/// <summary>
/// Two-Way-Actuator analog (mixing valve)
/// Zwei-Wege-Stellglied analog (Mischventil)
/// </summary>
FUNCTION_BLOCK PAEActuator2way_Analog EXTENDS PAEActuator1way_Analog
VAR_INPUT
	_IPos2 AT %I*: BOOL;	
END_VAR
VAR_OUTPUT
	_QPos2 AT %Q*: BOOL;	
END_VAR
VAR
	_PAPointMatIn2  : PAPoint(THIS^);
END_VAR

METHOD FB_init : BOOL
VAR_INPUT
	bInitRetains : BOOL; // if TRUE, the retain variables are initialized (warm start / cold start)
	bInCopyCode : BOOL;  // if TRUE, the instance afterwards gets moved into the copy code (online change)
	parent : IACComponent;
END_VAR
AddPoint(_PAPointMatIn1);
END_METHOD

METHOD PUBLIC HasPointReachedOffPosition : BOOL
VAR_INPUT
	point : IACPoint;
END_VAR
HasPointReachedOffPosition := SUPER^.HasPointReachedOffPosition(point);
END_METHOD

METHOD PUBLIC HasPointReachedOnPosition : BOOL
VAR_INPUT
	point : IACPoint;
END_VAR
HasPointReachedOnPosition := SUPER^.HasPointReachedOnPosition(point);
END_METHOD

PROPERTY PUBLIC PAPointMatIn2 : IACPoint
GET
PAPointMatIn2  := _PAPointMatIn2;
END_GET
END_PROPERTY

END_FUNCTION_BLOCK

(* stored: Version 1.1.0.1, ProductVersion 3.1.4020.12
   POU PAEActuator2way_Analog: Id {a2a041d8-6df1-467d-bb65-37358f54a768}, SpecialFunc None
   Method FB_init: Id {1a3bad42-9e08-41e2-b79f-a2631a4da060}
   Method HasPointReachedOffPosition: Id {2988950c-9b2f-409e-8f7a-84e8da5bc658}
   Method HasPointReachedOnPosition: Id {d2bade0b-1836-491f-896f-183f863eb4de}
   Property PAPointMatIn2: Id {901f576c-7f82-488b-915d-d8d590d987fb}
   Get Get: Id {d6a50b6e-fd2c-42fb-897e-f62f4197a367} *)
